// TIA Portal project "Proyecto2" (V16)

(* hardware
DEVICE "S7-1200 station_1"  S7-1200 Station
   slot 0: "Rack_0"  S7-1200 Rack  Rack  V1.0
   slot 1: "PLC_1"  CPU 1214C AC/DC/Rly  6ES7 214-1BG40-0XB0  V4.4
*)

// ===== PLC "PLC_1"  CPU 1214C AC/DC/Rly =====

VAR_GLOBAL   // PLC tag table "Tabla de variables estándar"
   "pulsador" AT %I0.0 : Bool;
   "motor" AT %Q0.0 : Bool;
   "pulsador_start" AT %I0.1 : Bool;
   "pulsador_stop" AT %I0.2 : Bool;
END_VAR

ORGANIZATION_BLOCK "Main"   // OB1, LAD, ProgramCycle
TITLE = "Main Program Sweep (Cycle)"
{ S7_Optimized_Access := 'TRUE' }
VERSION : 0.1
   VAR_INPUT
      Initial_Call : Bool;   // Initial call of this OB
      Remanence : Bool;   // =True, if remanent data are available
   END_VAR
BEGIN

REGION Network 1
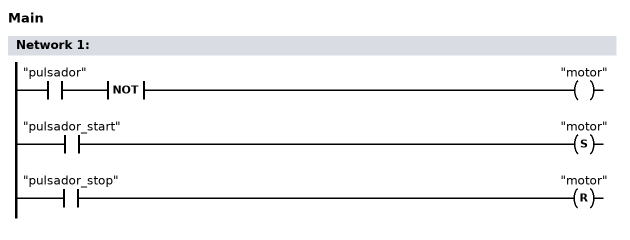
   RUNG wire#powerrail
      Contact( "pulsador" )
      Not()
      Coil( "motor" )
   END_RUNG
   RUNG wire#powerrail
      Contact( "pulsador_start" )
      S_Coil( "motor" )
   END_RUNG
   RUNG wire#powerrail
      Contact( "pulsador_stop" )
      R_Coil( "motor" )
   END_RUNG
   // the same network as SCL:
   "motor" := NOT "pulsador";
   IF "pulsador_start" THEN "motor" := TRUE; END_IF;
   IF "pulsador_stop" THEN "motor" := FALSE; END_IF;
END_REGION
END_ORGANIZATION_BLOCK